TYPE ST_MachineCommand :
	STRUCT
		LightOn : BOOL;
	END_STRUCT
END_TYPE

(* stored: Version 1.1.0.1, ProductVersion 3.1.4024.12
   DUT ST_MachineCommand: Id {843eab55-1788-46ac-a0f6-2e98ef8f65e5} *)
